INTERFACE I_CollectionNode EXTENDS I_Disposable

PROPERTY PUBLIC DataSize : UDINT
GET
END_GET
END_PROPERTY

METHOD PUBLIC Equals : BOOL
VAR_INPUT
	Symbol : ANY;
END_VAR
END_METHOD

METHOD PUBLIC TryGet : BOOL;
VAR_INPUT
	Destination : ANY;
END_VAR
END_METHOD

METHOD PUBLIC TryGetTo : BOOL;
VAR_INPUT
	DestinationAddress : PVOID;
	DestinationSize : UDINT;
END_VAR
END_METHOD

END_INTERFACE

(* stored: Version 1.1.0.1, ProductVersion 3.1.4024.12
   Itf I_CollectionNode: Id {5b4c873b-e072-47af-8e63-6d98eb3a2f02}
   Property DataSize: Id {18f9a4c9-70bc-4e4c-9f32-d840e79da13f}
   Get Get: Id {cfeb2235-325a-4950-ac6e-b849773697df}
   Method Equals: Id {a343db1e-bd0d-40a4-b217-2c35870d68a4}
   Method TryGet: Id {e3aaadc9-a69b-4db5-8f6e-b807b798613c}
   Method TryGetTo: Id {b3c69cd4-1eac-4cd3-a874-6b8d5dc47719} *)
